{library PUBLIC}
(*
 Status word for a specific device instance .
Function block DeviceUse or DeviceStatus will give you the status for a specific instance.
*)
TYPE INSTANCE_STATUS  : 
(
 	INSTANCE_STATUS_FREE:=0,							(* Instance not allocated *)
 	INSTANCE_STATUS_READY :=1,							(* Instance ready *)
 	INSTANCE_STATUS_BUSY:=2,							(* Instance is busy *)
	INSTANCE_STATUS_UNKNOWN:=3,							(* Unknown or address error *)

 	INSTANCE_STATUS_CANCEL:=-1							(* Instance cancel operation *)
);
END_TYPE
//  INSTANCE_STATUS_CANCEL = '-1'

(* stored: Version 1.1.0.1, ProductVersion 3.1.4024.2
   EnumerationTextList INSTANCE_STATUS: Id {7122a239-5cf8-428a-8a33-fae2a5f28592} *)
